// TIA Portal V19 export
TYPE "_AC_Interface"
   STRUCT
      ia : Struct   // Parameters ANY Pointer
         dbno : Int := 28;   // DB Number
         sta : Int;   // Starting Address (Byte offset)
         al : Int;   // Area Length in bytes
      END_STRUCT;
      IHW : HW_ANY;   // Device Hardware Identifier
      IIc : Int := -19456;   // I_CAP
      IIp : Int;   // IO-Link Master port the device is connected to
      op : Struct   // OP_interface ANY Pointer
         dbno : Int := 28;   // DB Number
         sta : Int;   // Starting Address (Byte offset)
         al : Int := 2;   // Area Length in bytes
      END_STRUCT;
      cmds : Struct   // Commands ANY Pointer
         dbno : Int := 28;   // DB Number
         sta : Int;   // Starting Address (Byte offset)
         al : Int := 4;   // Area Length in bytes
      END_STRUCT;
      ev : Struct   // Events ANY Pointer
         dbno : Int := 211;   // DB Number
         sta : Int;   // Starting Address (Byte offset)
         al : Int := 10;   // Area Length in bytes
      END_STRUCT;
      req : Struct   // ac/ev read/write request
         rd : Bool;   // ac read req
         wr : Bool;   // ac write req
         in : Bool;   // incoming Event
         out : Bool;   // outgoing Event
         cmd : Bool;   // command request
         spare : Bool;
         spare1 : Bool;
         spare2 : Bool;
         loaded : Bool;   // Event Request loaded for processing by _AC and or _EV
         VMrd : Bool;   // Valve Monitoring Read req
         VMrd_loaded : Bool;   // Valve Monitoring Read req loaded to FIFO
         FP : Bool;   // FP bit
         spare7 : Bool;
         spare8 : Bool;
         spare9 : Bool;
         spare10 : Bool;
      END_STRUCT;
   END_STRUCT;
END_TYPE
